Staubli VAL3: modbusSet.pgx

program modbusSet(num x_nNum (dimensions=1))
begin
  //通信正常，系统运行
  if (x_nNum==1)
    dStartState[0]=true
    dStartState[1]=false
    dStartState[2]=true
    dStartState[3]=false
    //通信正常，系统停止
  elseIf (x_nNum==2)
    dStartState[0]=true
    dStartState[1]=false
    dStartState[2]=false
    dStartState[3]=true
    //通信正常，系统复位
  elseIf (x_nNum==3)
    dStartState[0]=true
    dStartState[1]=true
    dStartState[2]=false
    dStartState[3]=false
    //0 通信准备，系统停止
  else
    dStartState[0]=true
    dStartState[1]=false
    dStartState[2]=false
    dStartState[3]=true
  endIf
end
